INTERFACE ITF_Cloneable

END_INTERFACE

(* stored: Version 1.1.0.1
   Itf ITF_Cloneable: Id {fb834b62-92a6-4712-860d-b7759ffea125} *)
